# EPICS autosave request: agilent53220/agilent53220_settings.req
$(P)$(Q):FREQ1:RBV.HIGH
$(P)$(Q):FREQ1:RBV.HIHI
$(P)$(Q):FREQ1:RBV.LOLO
$(P)$(Q):FREQ1:RBV.LOW
$(P)$(Q):FREQ2:RBV.HIGH
$(P)$(Q):FREQ2:RBV.HIHI
$(P)$(Q):FREQ2:RBV.LOLO
$(P)$(Q):FREQ2:RBV.LOW
$(P)$(Q):LEVEL1
$(P)$(Q):LEVEL2
$(P)$(Q):PHASE:RBV.HIGH
$(P)$(Q):PHASE:RBV.HIHI
$(P)$(Q):PHASE:RBV.LOLO
$(P)$(Q):PHASE:RBV.LOW
$(P)$(Q):UPDATE.SCAN
